(* IEC 61131-3 sources: SRCI/RobotLibrary/Library/POUs/Write/MC_WriteFrameData, 1 file *)

(* ---- MC_WriteFrameDataFB.st ---- *)
/// Change configuration of selected user frame number
FUNCTION_BLOCK MC_WriteFrameDataFB EXTENDS RobotLibraryBaseExecuteFB
// -------------------------------------------------------------------------
//  SRCI Robot Library
// -------------------------------------------------------------------------
//
//  Object:      WriteFrameDataFB
//  Author:      Thorsten Brach
//  Date:        2024-06-01
//
//  Description:
//
//
//  Copyright:
//    (C) 2024 Thorsten Brach. All rights reserved
//             Licensed under the LGPL-3.0 license.
//
//  Disclaimer:
//    This project is provided without any guarantee and can be used for
//    private and commercial purposes. Any use is at the user’s
//    own risk and responsibility.
//
// -------------------------------------------------------------------------
VAR_INPUT
  /// Processing Mode
  ProcessingMode     : ProcessingMode;
  /// Defines the target sequence in which the command will be executed
  SequenceFlag       : SequenceFlag;
  /// command parameter
  ParCmd             : WriteFrameDataParCmd;
END_VAR
VAR_OUTPUT
  /// Command is transferred and confirmed by the RC
  CommandBuffered    : BOOL;
  /// The command was aborted by another command
  CommandAborted     : BOOL;
  /// TRUE, while command is interrupted during execution and can be continued.
  CommandInterrupted : BOOL;
  /// command outputs
  OutCmd             : WriteFrameDataOutCmd;
END_VAR

VAR
  /// internal copy of command parameter
 _parCmd             : WriteFrameDataParCmd;
  /// command data to send
 _command            : WriteFrameDataSendData;
  /// response data received
 _response           : WriteFrameDataRecvData;
END_VAR

  SUPER^(AxesGroup := AxesGroup);

END_FUNCTION_BLOCK

METHOD INTERNAL CheckAddParameter : BOOL
VAR_INPUT
  /// Payload pointer
  PayloadPtr : UDINT;
END_VAR
VAR
  /// Payload as byte array
  Payload    : ARRAY [1..SIZEOF(_command)] OF BYTE;
  /// Null Byte array
  Null       : ARRAY [1..SIZEOF(_command)] OF BYTE;
  /// Data length to compare
  DataLen    : UDINT;
END_VAR

  // Payload pointer must be decreased by one byte, because ADR(Payload) is already one byte !
  PayloadPtr := LIMIT (0, PayloadPtr - 1, SIZEOF(Payload) -1);
  // Convert command struct to payload array
  SysDepMemCpy( pDest := ADR(Payload), pSrc := ADR(_command), DataLen := SIZEOF(_command));
  // Calculate the data length to compare - at least one byte must be compared !
  DataLen := LIMIT(1, SIZEOF(Payload) - PayloadPtr, SIZEOF(Payload));
  // Compare Payload-Array with Null-Byte-Array
  CheckAddParameter := SysDepMemCmp( pData1 := ADR(Payload) + PayloadPtr , pData2 := ADR(Null), DataLen := DataLen) <>  RobotLibraryConstants.OK ;

END_METHOD

METHOD PROTECTED CheckFunctionSupported : BOOL
VAR_IN_OUT
  /// Robot assignment of function
  AxesGroup : AxesGroup;
END_VAR

  CheckFunctionSupported := AxesGroup.State.RobotData.RCSupportedFunctions.WriteFrameData;

  IF ( NOT CheckFunctionSupported )
  THEN
    // call base implementation for set error and create log entry
    SUPER^.CheckFunctionSupported(AxesGroup := AxesGroup);
  END_IF

END_METHOD

METHOD PROTECTED CheckParameterChanged : BOOL
VAR_IN_OUT
  /// Robot assignment of function
  AxesGroup    : AxesGroup;
END_VAR

  // Check ParCmd Size is > 0, because MemCmp does not work correctly with size = 0
  IF (SIZEOF(ParCmd) = 0) OR (_stepCmd = 0)
  THEN
    RETURN;
  END_IF

  // compare memory
  _parameterChanged := ( SysDepMemCmp(pData1 := ADR(ParCmd), pData2 := ADR(_parCmd), DataLen := SIZEOF(ParCmd)) <> RobotLibraryConstants.OK );

  // check parameter valid ?
  _parameterValid   := CheckParameterValid( AxesGroup := AxesGroup );

  IF ((  _parameterChanged        )  AND
      (  _parameterValid          )) OR
      (  _parameterUpdateInternal )
  THEN
    // reset internal flag for send parameter update
   _parameterUpdateInternal := FALSE;
    // update internal copy of parameters
   _parCmd := ParCmd;
    // inc parameter sequence
   _command.ParSeq := _command.ParSeq + 1;
    // update command data
    CommandData := CreateCommandPayload(AxesGroup := AxesGroup); // ( Access via reference to rCommandFB in ACR )
    // notify active command register
    AxesGroup.Acyclic.ActiveCommandRegister.NotifyParameterChanged := _uniqueID;
  END_IF

END_METHOD

METHOD PROTECTED CheckParameterValid : BOOL
VAR_IN_OUT
  /// Robot assignment of function
  AxesGroup : AxesGroup;
END_VAR

  CheckParameterValid := TRUE;

  // Check ProcessingModea valid ?
  IF (( ProcessingMode <> ProcessingModeEnum.BUFFERED ) AND
      ( ProcessingMode <> ProcessingModeEnum.ABORTING ) AND
      ( ProcessingMode <> ProcessingModeEnum.PARALLEL ))
  THEN
    // Parameter not valid
    CheckParameterValid := FALSE;
    // Set error
    ErrorID := RobotLibraryErrorIdEnum.ERR_PROCESSINGMODE_NOT_ALLOWED;
    // Create log entry
    CreateLogMessagePara1 ( Timestamp   := AxesGroup.State.SystemTime,
                            MessageType := MessageType.CMD,
                            Severity    := Severity.ERROR,
                            MessageCode := ErrorID,
                            MessageText := 'Invalid Parameter ProcessingMode = {1}',
                            Para1       := PROCESSING_MODE_TO_STRING(ProcessingMode));
    RETURN;
  END_IF

  // Check SequenceFlag valid ?
  IF (( SequenceFlag <> SequenceFlagEnum.NO_SEQUENCE        ) AND
      ( SequenceFlag <> SequenceFlagEnum.PRIMARY_SEQUENCE   ) AND
      ( SequenceFlag <> SequenceFlagEnum.SECONDARY_SEQUENCE ))
  THEN
    // Parameter not valid
    CheckParameterValid := FALSE;
    // Set error
    ErrorID := RobotLibraryErrorIdEnum.ERR_SEQFLAG_NOT_ALLOWED;
    // Create log entry
    CreateLogMessagePara1 ( Timestamp   := AxesGroup.State.SystemTime,
                            MessageType := MessageType.CMD,
                            Severity    := Severity.ERROR,
                            MessageCode := ErrorID,
                            MessageText := 'Invalid Parameter SequenceFlag = {1}',
                            Para1       := SEQUENCE_FLAG_TO_STRING(SequenceFlag));
    RETURN;
  END_IF

  // Check ParCmd.FrameNo valid ?
  IF (( ParCmd.FrameNo < 0                                                   ) OR
      ( ParCmd.FrameNo > 254                                                 ) OR
      ( ParCmd.FrameNo > AxesGroup.State.ConfigurationData.HighestFrameIndex ) OR
      ( ParCmd.FrameNo > RobotLibraryParameter.FRAME_MAX -1                  ))
  THEN
    // Parameter not valid
    CheckParameterValid := FALSE;

    // Check FrameNo available on RC ?
    IF ( ParCmd.FrameNo > AxesGroup.State.ConfigurationData.HighestFrameIndex )
    THEN
      ErrorID := RobotLibraryErrorIdEnum.ERR_FRAMENO_UNAVAILABLE;
    ELSE
      ErrorID := RobotLibraryErrorIdEnum.ERR_FRAMENO_RANGE;
  	END_IF

    // Create log entry
    CreateLogMessagePara1 ( Timestamp   := AxesGroup.State.SystemTime,
                            MessageType := MessageType.CMD,
                            Severity    := Severity.ERROR,
                            MessageCode := ErrorID,
                            MessageText := 'Invalid Parameter ParCmd.FrameNo = {1}',
                            Para1       := USINT_TO_STRING(ParCmd.FrameNo));
    RETURN;
  END_IF

  // Check ParCmd.FrameData.ReferenceFrame valid ?
  IF (( ParCmd.FrameData.ReferenceFrame < 0   ) OR
      ( ParCmd.FrameData.ReferenceFrame > 254 ))
  THEN
    // Parameter not valid
    CheckParameterValid := FALSE;
    // Set error
    ErrorID := RobotLibraryErrorIdEnum.ERR_INVALID_PAR_CMD;
    // Create log entry
    CreateLogMessagePara1 ( Timestamp   := AxesGroup.State.SystemTime,
                            MessageType := MessageType.CMD,
                            Severity    := Severity.ERROR,
                            MessageCode := ErrorID,
                            MessageText := 'Invalid Parameter ParCmd.FrameData.ReferenceFrame = {1}',
                            Para1       := USINT_TO_STRING(ParCmd.FrameData.ReferenceFrame));
    RETURN;
  END_IF

  // Check ParCmd.FrameData.X ?
  IF ( SysDepIsValidReal(ParCmd.FrameData.X) = FALSE )
  THEN
    // Parameter not valid
    CheckParameterValid := FALSE;
    // Set error
    ErrorID := RobotLibraryErrorIdEnum.ERR_INVALID_PAR_CMD;

    // Create log entry
    CreateLogMessagePara1 ( Timestamp   := AxesGroup.State.SystemTime,
                            MessageType := MessageType.CMD,
                            Severity    := Severity.ERROR,
                            MessageCode := ErrorID,
                            MessageText := 'Invalid Parameter ParCmd.FrameData.X = {1}',
                            Para1       := VALID_REAL_TO_STRING(ParCmd.FrameData.X));
    RETURN;
  END_IF

  // Check ParCmd.FrameData.Y ?
  IF ( SysDepIsValidReal(ParCmd.FrameData.Y) = FALSE )
  THEN
    // Parameter not valid
    CheckParameterValid := FALSE;
    // Set error
    ErrorID := RobotLibraryErrorIdEnum.ERR_INVALID_PAR_CMD;

    // Create log entry
    CreateLogMessagePara1 ( Timestamp   := AxesGroup.State.SystemTime,
                            MessageType := MessageType.CMD,
                            Severity    := Severity.ERROR,
                            MessageCode := ErrorID,
                            MessageText := 'Invalid Parameter ParCmd.FrameData.Y = {1}',
                            Para1       := VALID_REAL_TO_STRING(ParCmd.FrameData.Y));
    RETURN;
  END_IF

  // Check ParCmd.FrameData.Z ?
  IF ( SysDepIsValidReal(ParCmd.FrameData.Z) = FALSE )
  THEN
    // Parameter not valid
    CheckParameterValid := FALSE;
    // Set error
    ErrorID := RobotLibraryErrorIdEnum.ERR_INVALID_PAR_CMD;

    // Create log entry
    CreateLogMessagePara1 ( Timestamp   := AxesGroup.State.SystemTime,
                            MessageType := MessageType.CMD,
                            Severity    := Severity.ERROR,
                            MessageCode := ErrorID,
                            MessageText := 'Invalid Parameter ParCmd.FrameData.Z = {1}',
                            Para1       := VALID_REAL_TO_STRING(ParCmd.FrameData.Z));
    RETURN;
  END_IF

  // Check ParCmd.FrameData.Rx ?
  IF ( SysDepIsValidReal(ParCmd.FrameData.Rx) = FALSE )
  THEN
    // Parameter not valid
    CheckParameterValid := FALSE;
    // Set error
    ErrorID := RobotLibraryErrorIdEnum.ERR_INVALID_PAR_CMD;

    // Create log entry
    CreateLogMessagePara1 ( Timestamp   := AxesGroup.State.SystemTime,
                            MessageType := MessageType.CMD,
                            Severity    := Severity.ERROR,
                            MessageCode := ErrorID,
                            MessageText := 'Invalid Parameter ParCmd.FrameData.Rx = {1}',
                            Para1       := VALID_REAL_TO_STRING(ParCmd.FrameData.Rx));
    RETURN;
  END_IF

  // Check ParCmd.FrameData.Ry ?
  IF ( SysDepIsValidReal(ParCmd.FrameData.Ry) = FALSE )
  THEN
    // Parameter not valid
    CheckParameterValid := FALSE;
    // Set error
    ErrorID := RobotLibraryErrorIdEnum.ERR_INVALID_PAR_CMD;

    // Create log entry
    CreateLogMessagePara1 ( Timestamp   := AxesGroup.State.SystemTime,
                            MessageType := MessageType.CMD,
                            Severity    := Severity.ERROR,
                            MessageCode := ErrorID,
                            MessageText := 'Invalid Parameter ParCmd.FrameData.Ry = {1}',
                            Para1       := VALID_REAL_TO_STRING(ParCmd.FrameData.Ry));
    RETURN;
  END_IF

  // Check ParCmd.FrameData.Rz ?
  IF ( SysDepIsValidReal(ParCmd.FrameData.Rz) = FALSE )
  THEN
    // Parameter not valid
    CheckParameterValid := FALSE;
    // Set error
    ErrorID := RobotLibraryErrorIdEnum.ERR_INVALID_PAR_CMD;

    // Create log entry
    CreateLogMessagePara1 ( Timestamp   := AxesGroup.State.SystemTime,
                            MessageType := MessageType.CMD,
                            Severity    := Severity.ERROR,
                            MessageCode := ErrorID,
                            MessageText := 'Invalid Parameter ParCmd.FrameData.Rz = {1}',
                            Para1       := VALID_REAL_TO_STRING(ParCmd.FrameData.Rz));
    RETURN;
  END_IF

END_METHOD

METHOD INTERNAL CreateCommandPayload : RobotLibraryCommandDataFB
VAR_IN_OUT
  /// Robot assignment of function
  AxesGroup : AxesGroup;
END_VAR
VAR
  /// Parameter count
 _parameterCnt : DINT;
END_VAR
// Table 6-120: Sent CMD payload (PLC to RC) of "WriteFrameData"
// --------------------------
// Header
// --------------------------
// Byte 00 : UINT  - Type HB
// Byte 01 :       - Type LB
// Byte 02 : USINT - Reserve | ExecutionMode
// Byte 03 : USINT - ParSeq  | Priority
// --------------------------
// Datablock
// --------------------------
// Byte 04 : DATE FrameData.Date
// Byte 05 :
// Byte 06 : TIME_OF_DAY FrameData.Time
// Byte 07 :
// Byte 08 :
// Byte 09 :
// Byte 10 : USINT FrameData.ReferenceFrame
// Byte 11 : BYTE Reserved
// Byte 12 : REAL FrameData.X
// Byte 13 :
// Byte 14 :
// Byte 15 :
// Byte 16 : REAL FrameData.Y
// Byte 17 :
// Byte 18 :
// Byte 19 :
// Byte 20 : REAL FrameData.Z
// Byte 21 :
// Byte 22 :
// Byte 23 :
// Byte 24 : REAL FrameData.RX
// Byte 25 :
// Byte 26 :
// Byte 27 :
// Byte 28 : REAL FrameData.RY
// Byte 29 :
// Byte 30 :
// Byte 31 :
// Byte 32 : REAL FrameData.RZ
// Byte 33 :
// Byte 34 :
// Byte 35 :
// Byte 36 : USINT FrameNo
// --------------------------

  // set command parameter
  _command.CmdTyp    :=  CmdType.WriteFrameData;
  _command.ExecMode  :=  ExecMode;
  _command.ParSeq    := _command.ParSeq;
  _command.Priority  :=  Priority;
  _command.Reserve   := 0;
  _command.FrameData := _parCmd.FrameData;
  _command.FrameNo   := _parCmd.FrameNo;

  // copy command data to header
  _cmdHeader := _command;
  // call base implementation to copy header to payload buffer
  CreateCommandPayload := SUPER^.CreateCommandPayload(AxesGroup := AxesGroup);

  // Check parameter must be added ?
  IF ( CheckAddParameter(CreateCommandPayload.PayloadPtr))
  THEN
    // add command.FrameData.Timestamp.IEC_DATE
    CreateCommandPayload.AddUint(_command.FrameData.Timestamp.IEC_DATE);
    // inc parameter counter
   _parameterCnt := _parameterCnt + 1;
  END_IF

  // Check parameter must be added ?
  IF ( CheckAddParameter(CreateCommandPayload.PayloadPtr))
  THEN
    // add command.FrameData.Timestamp.IEC_TIME
    CreateCommandPayload.AddTime(_command.FrameData.Timestamp.IEC_TIME);
    // inc parameter counter
   _parameterCnt := _parameterCnt + 1;
  END_IF

  // Check parameter must be added ?
  IF ( CheckAddParameter(CreateCommandPayload.PayloadPtr))
  THEN
    // add command.FrameData.ReferenceFrame
    CreateCommandPayload.AddUsint(_command.FrameData.ReferenceFrame);
    // inc parameter counter
   _parameterCnt := _parameterCnt + 1;
  END_IF

  // Check parameter must be added ?
  IF ( CheckAddParameter(CreateCommandPayload.PayloadPtr))
  THEN
    // add command.Reserver
    CreateCommandPayload.AddByte(_command.Reserve);
    // inc parameter counter
   _parameterCnt := _parameterCnt + 1;
  END_IF

  // Check parameter must be added ?
  IF ( CheckAddParameter(CreateCommandPayload.PayloadPtr))
  THEN
    // add command.FrameData.X
    CreateCommandPayload.AddReal(_command.FrameData.X);
    // inc parameter counter
   _parameterCnt := _parameterCnt + 1;
  END_IF

  // Check parameter must be added ?
  IF ( CheckAddParameter(CreateCommandPayload.PayloadPtr))
  THEN
    // add command.FrameData.Y
    CreateCommandPayload.AddReal(_command.FrameData.Y);
    // inc parameter counter
   _parameterCnt := _parameterCnt + 1;
  END_IF

  // Check parameter must be added ?
  IF ( CheckAddParameter(CreateCommandPayload.PayloadPtr))
  THEN
    // add command.FrameData.Z
    CreateCommandPayload.AddReal(_command.FrameData.Z);
    // inc parameter counter
   _parameterCnt := _parameterCnt + 1;
  END_IF

  // Check parameter must be added ?
  IF ( CheckAddParameter(CreateCommandPayload.PayloadPtr))
  THEN
    // add command.FrameData.Rx
    CreateCommandPayload.AddReal(_command.FrameData.Rx);
    // inc parameter counter
   _parameterCnt := _parameterCnt + 1;
  END_IF

  // Check parameter must be added ?
  IF ( CheckAddParameter(CreateCommandPayload.PayloadPtr))
  THEN
    // add command.FrameData.Ry
    CreateCommandPayload.AddReal(_command.FrameData.Ry);
    // inc parameter counter
   _parameterCnt := _parameterCnt + 1;
  END_IF

  // Check parameter must be added ?
  IF ( CheckAddParameter(CreateCommandPayload.PayloadPtr))
  THEN
    // add command.FrameData.Rz
    CreateCommandPayload.AddReal(_command.FrameData.Rz);
    // inc parameter counter
   _parameterCnt := _parameterCnt + 1;
  END_IF

  // Check parameter must be added ?
  IF ( CheckAddParameter(CreateCommandPayload.PayloadPtr))
  THEN
    // add command.FrameNo
    CreateCommandPayload.AddUsint(_command.FrameNo);
    // inc parameter counter
   _parameterCnt := _parameterCnt + 1;
  END_IF

  // Create logging
  CreateCommandPayloadLog(AxesGroup := AxesGroup, ParameterCnt := _parameterCnt);

END_METHOD

METHOD INTERNAL CreateCommandPayloadLog
VAR_IN_OUT
  /// Robot assignment of function
  AxesGroup : AxesGroup;
END_VAR
VAR_INPUT
  /// Parameter count
  ParameterCnt : DINT;
END_VAR

  // Create log entry for Parameter start
  CreateLogMessagePara1 ( Timestamp   := AxesGroup.State.SystemTime,
                          MessageType := MessageType.CMD,
                          Severity    := Severity.DEBUG,
                          MessageCode := 0,
                          MessageText := 'Create command payload with the {1} parameter(s) :',
                          Para1       := DINT_TO_STRING(ParameterCnt));

  // Return if no parameter is remaining...
  IF ( ParameterCnt = 0 ) THEN RETURN; END_IF
  // dec remaining parameter(s)
  ParameterCnt := ParameterCnt - 1;
  // Create log entry for FrameData.Timestamp.IEC_DATE
  CreateLogMessagePara1 ( Timestamp   := AxesGroup.State.SystemTime,
                          MessageType := MessageType.CMD,
                          Severity    := Severity.DEBUG,
                          MessageCode := 0,
                          MessageText := 'Command.FrameData.Timestamp.IEC_DATE = {1}',
                          Para1       :=  IEC_DATE_TO_STRING(_command.FrameData.Timestamp.IEC_DATE));

  // Return if no parameter is remaining...
  IF ( ParameterCnt = 0 ) THEN RETURN; END_IF
  // dec remaining parameter(s)
  ParameterCnt := ParameterCnt - 1;
  // Create log entry for FrameData.Timestamp.IEC_TIME
  CreateLogMessagePara1 ( Timestamp   := AxesGroup.State.SystemTime,
                          MessageType := MessageType.CMD,
                          Severity    := Severity.DEBUG,
                          MessageCode := 0,
                          MessageText := 'Command.FrameData.Timestamp.IEC_TIME = {1}',
                          Para1       :=  IEC_TIME_TO_STRING(_command.FrameData.Timestamp.IEC_TIME));

  // Return if no parameter is remaining...
  IF ( ParameterCnt = 0 ) THEN RETURN; END_IF
  // dec remaining parameter(s)
  ParameterCnt := ParameterCnt - 1;
  // Create log entry for FrameData.ReferenceFrame
  CreateLogMessagePara1 ( Timestamp   := AxesGroup.State.SystemTime,
                          MessageType := MessageType.CMD,
                          Severity    := Severity.DEBUG,
                          MessageCode := 0,
                          MessageText := 'Command.FrameData.ReferenceFrame = {1}',
                          Para1       :=  USINT_TO_STRING(_command.FrameData.ReferenceFrame));

  // Return if no parameter is remaining...
  IF ( ParameterCnt = 0 ) THEN RETURN; END_IF
  // dec remaining parameter(s)
  ParameterCnt := ParameterCnt - 1;
  // Create log entry for Reserve
  CreateLogMessagePara1 ( Timestamp   := AxesGroup.State.SystemTime,
                          MessageType := MessageType.CMD,
                          Severity    := Severity.DEBUG,
                          MessageCode := 0,
                          MessageText := 'Command.Reserve = {1}',
                          Para1       :=  BYTE_TO_STRING(_command.Reserve));

  // Return if no parameter is remaining...
  IF ( ParameterCnt = 0 ) THEN RETURN; END_IF
  // dec remaining parameter(s)
  ParameterCnt := ParameterCnt - 1;
  // Create log entry for FrameData.X
  CreateLogMessagePara1 ( Timestamp   := AxesGroup.State.SystemTime,
                          MessageType := MessageType.CMD,
                          Severity    := Severity.DEBUG,
                          MessageCode := 0,
                          MessageText := 'Command.FrameData.X = {1}',
                          Para1       :=  REAL_TO_STRING(_command.FrameData.X));

  // Return if no parameter is remaining...
  IF ( ParameterCnt = 0 ) THEN RETURN; END_IF
  // dec remaining parameter(s)
  ParameterCnt := ParameterCnt - 1;
  // Create log entry for FrameData.Y
  CreateLogMessagePara1 ( Timestamp   := AxesGroup.State.SystemTime,
                          MessageType := MessageType.CMD,
                          Severity    := Severity.DEBUG,
                          MessageCode := 0,
                          MessageText := 'Command.FrameData.Y = {1}',
                          Para1       :=  REAL_TO_STRING(_command.FrameData.Y));

  // Return if no parameter is remaining...
  IF ( ParameterCnt = 0 ) THEN RETURN; END_IF
  // dec remaining parameter(s)
  ParameterCnt := ParameterCnt - 1;
  // Create log entry for FrameData.Z
  CreateLogMessagePara1 ( Timestamp   := AxesGroup.State.SystemTime,
                          MessageType := MessageType.CMD,
                          Severity    := Severity.DEBUG,
                          MessageCode := 0,
                          MessageText := 'Command.FrameData.Z = {1}',
                          Para1       :=  REAL_TO_STRING(_command.FrameData.Z));

  // Return if no parameter is remaining...
  IF ( ParameterCnt = 0 ) THEN RETURN; END_IF
  // dec remaining parameter(s)
  ParameterCnt := ParameterCnt - 1;
  // Create log entry for FrameData.Rx
  CreateLogMessagePara1 ( Timestamp   := AxesGroup.State.SystemTime,
                          MessageType := MessageType.CMD,
                          Severity    := Severity.DEBUG,
                          MessageCode := 0,
                          MessageText := 'Command.FrameData.Rx = {1}',
                          Para1       :=  REAL_TO_STRING(_command.FrameData.Rx));

  // Return if no parameter is remaining...
  IF ( ParameterCnt = 0 ) THEN RETURN; END_IF
  // dec remaining parameter(s)
  ParameterCnt := ParameterCnt - 1;
  // Create log entry for FrameData.Ry
  CreateLogMessagePara1 ( Timestamp   := AxesGroup.State.SystemTime,
                          MessageType := MessageType.CMD,
                          Severity    := Severity.DEBUG,
                          MessageCode := 0,
                          MessageText := 'Command.FrameData.Ry = {1}',
                          Para1       :=  REAL_TO_STRING(_command.FrameData.Ry));

  // Return if no parameter is remaining...
  IF ( ParameterCnt = 0 ) THEN RETURN; END_IF
  // dec remaining parameter(s)
  ParameterCnt := ParameterCnt - 1;
  // Create log entry for FrameData.Rz
  CreateLogMessagePara1 ( Timestamp   := AxesGroup.State.SystemTime,
                          MessageType := MessageType.CMD,
                          Severity    := Severity.DEBUG,
                          MessageCode := 0,
                          MessageText := 'Command.FrameData.Rz = {1}',
                          Para1       :=  REAL_TO_STRING(_command.FrameData.Rz));

  // Return if no parameter is remaining...
  IF ( ParameterCnt = 0 ) THEN RETURN; END_IF
  // dec remaining parameter(s)
  ParameterCnt := ParameterCnt - 1;
  // Create log entry for FrameNo
  CreateLogMessagePara1 ( Timestamp   := AxesGroup.State.SystemTime,
                          MessageType := MessageType.CMD,
                          Severity    := Severity.DEBUG,
                          MessageCode := 0,
                          MessageText := 'Command.FrameNo = {1}',
                          Para1       :=  USINT_TO_STRING(_command.FrameNo));

END_METHOD

METHOD FB_init : BOOL
VAR_INPUT
  /// if TRUE, the retain variables are initialized (warm start / cold start)
  bInitRetains : BOOL;
  /// if TRUE, the instance afterwards gets moved into the copy code (online change)
  bInCopyCode  : BOOL;
END_VAR

  MyType := 'MC_WriteFrameDataFB';

  ExecMode       := ExecutionMode.PARALLEL;
  Priority       := PriorityLevel.NORMAL;
  ProcessingMode := ProcessingModeEnum.PARALLEL;
  SequenceFlag   := SequenceFlagEnum.NO_SEQUENCE;

END_METHOD

METHOD PROTECTED OnExecRun : DINT
VAR_IN_OUT
  /// Robot assignment of function
  AxesGroup : AxesGroup;
END_VAR

  // call base implementation
  SUPER^.OnExecRun(AxesGroup := AxesGroup);

  CASE _stepCmd OF

    00:  IF ( _execute_R.Q ) AND ( NOT Error)
         THEN
           // Check function is supported and parameter are valid ?
           IF (( CheckFunctionSupported( AxesGroup := AxesGroup )) AND
               ( CheckParameterValid   ( AxesGroup := AxesGroup )))
           THEN
             // set busy flag
             Busy := TRUE;
             // Reset command outputs
             SysDepMemSet(pDest := ADR(OutCmd), Value := 0, DataLen := SIZEOF(OutCmd));
             // apply command parameter
            _parCmd := ParCmd;
             // init parameter sequence
            _command.ParSeq := 1;
             // create command data
             CommandData := CreateCommandPayload(AxesGroup := AxesGroup);
             // Add command to active command register
            _uniqueID := AxesGroup.Acyclic.ActiveCommandRegister.AddCmd( pCommandFB := ADR(THIS^ ));
             // set timeout
             SetTimeout(PT := _timeoutCmd, rTimer := _timerCmd);
             // inc step counter
            _stepCmd := _stepCmd + 1;
           END_IF
         END_IF

    01:  // Wait for responce received
         IF ( _responseReceived )
         THEN
           // reset response received flag
          _responseReceived := FALSE;

           CASE  _response.State
           OF
             CmdMessageState.BUFFERED    : CommandBuffered    := TRUE;
             CmdMessageState.ABORTED     : CommandAborted     := TRUE;
             CmdMessageState.INTERRUPTED : CommandInterrupted := TRUE;
             CmdMessageState.DONE        : Done               := TRUE;
             CmdMessageState.ERROR       : Error              := TRUE;
           END_CASE

           // Done, Aborted or Error ?
           IF (_response.State >= CmdMessageState.DONE )
           THEN
             // Reset Busy flag
             Busy := FALSE;
             // set timeout
             SetTimeout(PT := _timeoutCmd, rTimer := _timerCmd);
             // inc step counter
            _stepCmd := _stepCmd + 1;
           END_IF
         END_IF

    02: IF ( NOT Execute)
        THEN
          Reset();
        END_IF

  ELSE
    // invalid step
    ErrorID := RobotLibraryErrorIdEnum.ERR_INVALID_STEP;
  END_CASE

  // Reset FB
  IF ( NOT Execute )
  THEN
    Reset();
  END_IF

END_METHOD

METHOD INTERNAL ParseResponsePayload : DINT
VAR_INPUT
  /// Response data
  ResponseData : RobotLibraryResponseDataFB;
  /// Timestamp
  Timestamp    : SystemTime;
END_VAR
VAR
  /// Parameter count
 _parameterCnt : DINT;
END_VAR
// Table 6-121: Received CMD payload (RC to PLC) of "WriteFrameData"
// --------------------------
// Header
// --------------------------
// Byte 00 : USINT   - ParSeq | State
// Byte 01 : SINT    - AlarmMessageSeverity
// Byte 02 : UINT    - AlarmMessageCode HB
// Byte 03 :         - AlarmMessageCode LB
// --------------------------
// Datablock
// --------------------------
// Byte 04 : USINT      - InvocationCounter
// Byte 05 : SINT       - Reserved
// Byte 06 : INT        - OriginID HW HB
// Byte 07 :            - OriginID HW LB

  // call base implementation to parse the header from payload buffer
  ResponseData.PayloadPtr := SUPER^.ParseResponsePayload(ResponseData := ResponseData, Timestamp := Timestamp);

  // copy parsed header to response
  _response.ParSeq               := _rspHeader.ParSeq;
  _response.State                := _rspHeader.State;
  _response.AlarmMessageSeverity := _rspHeader.AlarmMessageSeverity;
  _response.AlarmMessageCode     := _rspHeader.AlarmMessageCode;

  // Create logging
  ParseResponsePayloadLog(ResponseData := ResponseData, Timestamp := Timestamp, ParameterCnt := _parameterCnt);

END_METHOD

METHOD INTERNAL ParseResponsePayloadLog
VAR_INPUT
  /// Response data
  ResponseData : RobotLibraryResponseDataFB;
  /// Timestamp
  Timestamp    : SystemTime;
  /// Parameter count
  ParameterCnt : DINT;
END_VAR

  // Create log entry for Parameter start
  CreateLogMessagePara1 ( Timestamp   := Timestamp,
                          MessageType := MessageType.CMD,
                          Severity    := Severity.DEBUG,
                          MessageCode := 0,
                          MessageText := '{1} parameter(s) to parse from the response data:',
                          Para1       := DINT_TO_STRING(ParameterCnt));

  // Return if no parameter is remaining...
  IF ( ParameterCnt = 0 ) THEN RETURN; END_IF
  // dec remaining parameter(s)
  ParameterCnt := ParameterCnt - 1;
  // Create log entry for no parameter
  CreateLogMessage      ( Timestamp   := Timestamp,
                          MessageType := MessageType.CMD,
                          Severity    := Severity.DEBUG,
                          MessageCode := 0,
                          MessageText := 'This command has no parameter to parse...');

END_METHOD

METHOD PROTECTED Reset : DINT
VAR_INPUT
END_VAR

  Reset := SUPER^.Reset();

  Done               := FALSE;
  Busy               := FALSE;
  CommandBuffered    := FALSE;
  CommandAborted     := FALSE;
  CommandInterrupted := FALSE;

END_METHOD
